FUNCTION_BLOCK TestBoolAdapter (* Template for an empty basic function block *)
  (* Standard: 61499-2; Description: Copyright (c) 2019 Jan Holzweber This program and the accompanying materials are made available under the terms of the Eclipse Public License 2.0 which is available at https://www.eclipse.org/legal/epl-2.0/ SPDX-License-Identifier: EPL-2.0 *)
  (* Version 1.0, 2019-07-18, Jan Holzweber *)
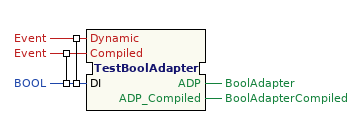
  EVENT_INPUT
    Dynamic WITH DI;
    Compiled WITH DI;
  END_EVENT
  VAR_INPUT
    DI : BOOL;
  END_VAR
  PLUGS
    ADP : BoolAdapter;
    ADP_Compiled : BoolAdapterCompiled;
  END_PLUGS
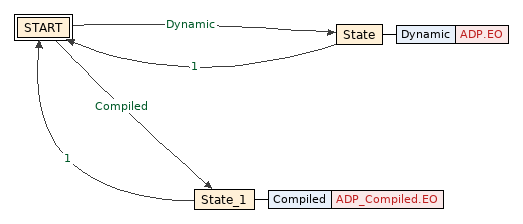
  EC_STATES
    START; (* Initial State *)
    State : Dynamic -> ADP.EO;
    State_1 : Compiled -> ADP_Compiled.EO;
  END_STATES
  EC_TRANSITIONS
    START TO State := Dynamic;
    State TO START := 1;
    START TO State_1 := Compiled;
    State_1 TO START := 1;
  END_TRANSITIONS
  ALGORITHM Dynamic IN ST: (* new algorithm *)
ADP.BO := DI;
  END_ALGORITHM
  ALGORITHM Compiled IN ST: (* new algorithm *)
ADP_Compiled.BO := DI;
  END_ALGORITHM
END_FUNCTION_BLOCK
